// Mitsubishi GX Works2 project: Conveyor   PLC: Q03UD

PROGRAM IOCHECK
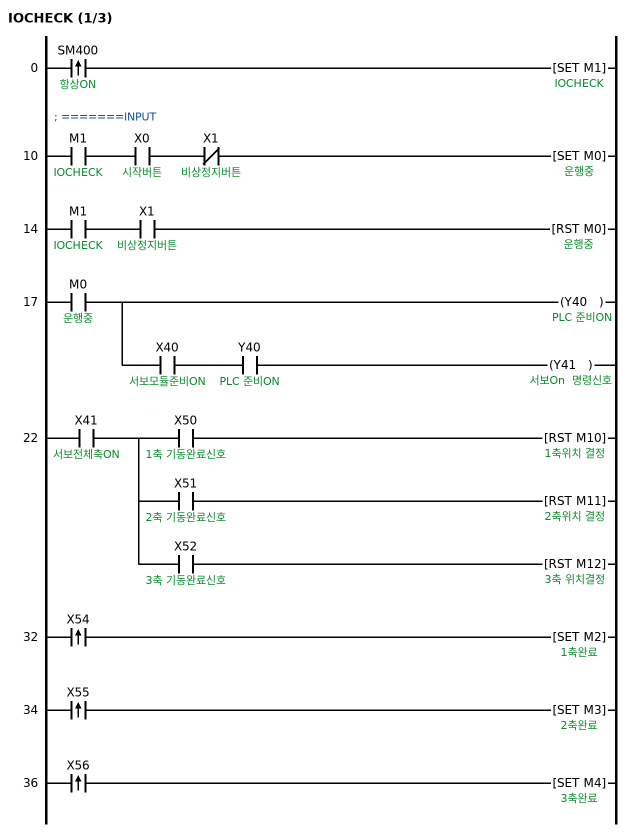
0     LDP     SM400  ; 항상ON
      SET     M1  ; IOCHECK
; =======INPUT
10    LD      M1  ; IOCHECK
      AND     X0  ; 시작버튼
      ANI     X1  ; 비상정지버튼
      SET     M0  ; 운행중
14    LD      M1  ; IOCHECK
      AND     X1  ; 비상정지버튼
      RST     M0  ; 운행중
17    LD      M0  ; 운행중
      OUT     Y40  ; PLC 준비ON
      AND     X40  ; 서보모듈준비ON
      AND     Y40  ; PLC 준비ON
      OUT     Y41  ; 서보On  명령신호
22    LD      X41  ; 서보전체축ON
      MPS
      AND     X50  ; 1축 기동완료신호
      RST     M10  ; 1축위치 결정
      MRD
      AND     X51  ; 2축 기동완료신호
      RST     M11  ; 2축위치 결정
      MPP
      AND     X52  ; 3축 기동완료신호
      RST     M12  ; 3축 위치결정
32    LDP     X54
      SET     M2  ; 1축완료
34    LDP     X55
      SET     M3  ; 2축완료
36    LDP     X56
      SET     M4  ; 3축완료
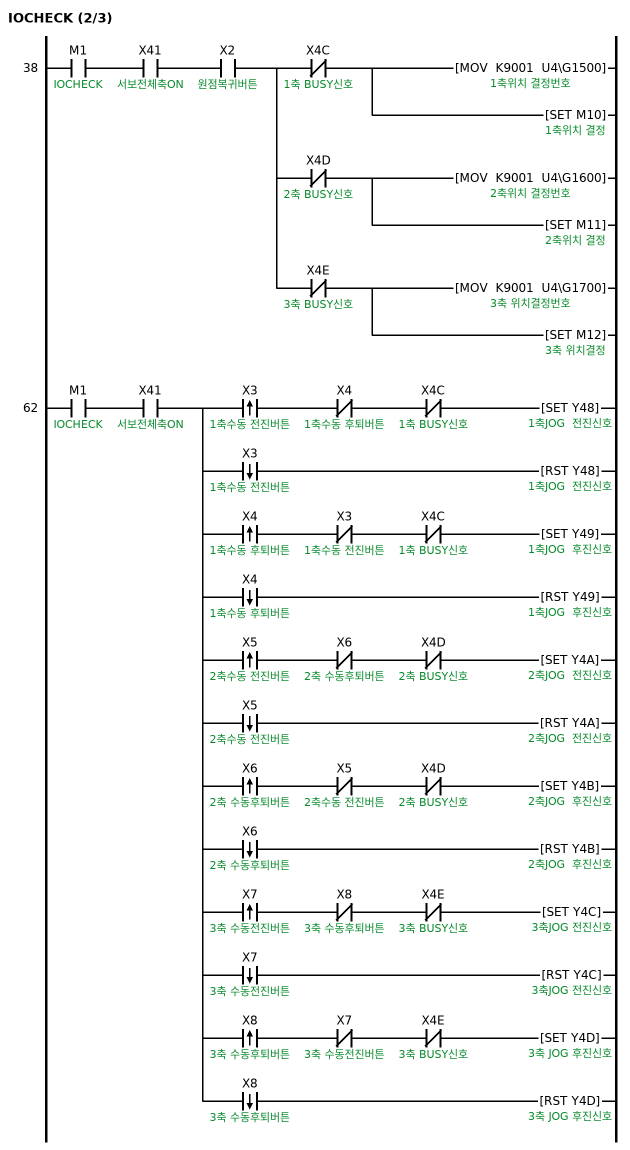
38    LD      M1  ; IOCHECK
      AND     X41  ; 서보전체축ON
      AND     X2  ; 원점복귀버튼
      MPS
      ANI     X4C  ; 1축 BUSY신호
      MOV     K9001 U4\G1500  ; 1축위치 결정번호
      SET     M10  ; 1축위치 결정
      MRD
      ANI     X4D  ; 2축 BUSY신호
      MOV     K9001 U4\G1600  ; 2축위치 결정번호
      SET     M11  ; 2축위치 결정
      MPP
      ANI     X4E  ; 3축 BUSY신호
      MOV     K9001 U4\G1700  ; 3축 위치결정번호
      SET     M12  ; 3축 위치결정
62    LD      M1  ; IOCHECK
      AND     X41  ; 서보전체축ON
      MPS
      ANDP    X3  ; 1축수동 전진버튼
      ANI     X4  ; 1축수동 후퇴버튼
      ANI     X4C  ; 1축 BUSY신호
      SET     Y48  ; 1축JOG  전진신호
      MRD
      ANDF    X3  ; 1축수동 전진버튼
      RST     Y48  ; 1축JOG  전진신호
      MRD
      ANDP    X4  ; 1축수동 후퇴버튼
      ANI     X3  ; 1축수동 전진버튼
      ANI     X4C  ; 1축 BUSY신호
      SET     Y49  ; 1축JOG  후진신호
      MRD
      ANDF    X4  ; 1축수동 후퇴버튼
      RST     Y49  ; 1축JOG  후진신호
      MRD
      ANDP    X5  ; 2축수동 전진버튼
      ANI     X6  ; 2축 수동후퇴버튼
      ANI     X4D  ; 2축 BUSY신호
      SET     Y4A  ; 2축JOG  전진신호
      MRD
      ANDF    X5  ; 2축수동 전진버튼
      RST     Y4A  ; 2축JOG  전진신호
      MRD
      ANDP    X6  ; 2축 수동후퇴버튼
      ANI     X5  ; 2축수동 전진버튼
      ANI     X4D  ; 2축 BUSY신호
      SET     Y4B  ; 2축JOG  후진신호
      MRD
      ANDF    X6  ; 2축 수동후퇴버튼
      RST     Y4B  ; 2축JOG  후진신호
      MRD
      ANDP    X7  ; 3축 수동전진버튼
      ANI     X8  ; 3축 수동후퇴버튼
      ANI     X4E  ; 3축 BUSY신호
      SET     Y4C  ; 3축JOG 전진신호
      MRD
      ANDF    X7  ; 3축 수동전진버튼
      RST     Y4C  ; 3축JOG 전진신호
      MRD
      ANDP    X8  ; 3축 수동후퇴버튼
      ANI     X7  ; 3축 수동전진버튼
      ANI     X4E  ; 3축 BUSY신호
      SET     Y4D  ; 3축 JOG 후진신호
      MPP
      ANDF    X8  ; 3축 수동후퇴버튼
      RST     Y4D  ; 3축 JOG 후진신호
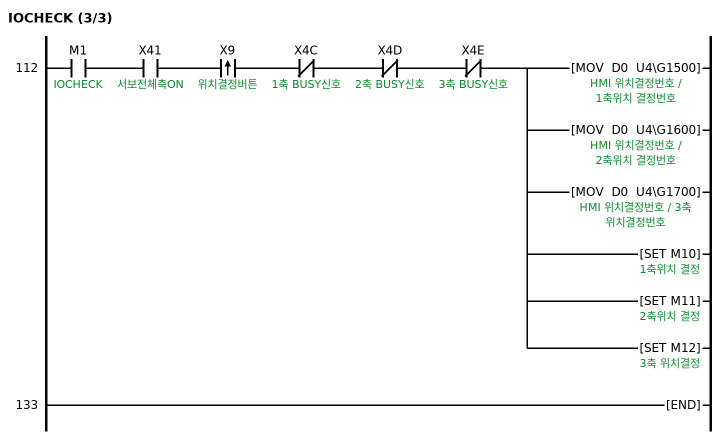
112   LD      M1  ; IOCHECK
      AND     X41  ; 서보전체축ON
      ANDP    X9  ; 위치결정버튼
      ANI     X4C  ; 1축 BUSY신호
      ANI     X4D  ; 2축 BUSY신호
      ANI     X4E  ; 3축 BUSY신호
      MOV     D0 U4\G1500  ; HMI 위치결정번호
      MOV     D0 U4\G1600
      MOV     D0 U4\G1700
      SET     M10  ; 1축위치 결정
      SET     M11  ; 2축위치 결정
      SET     M12  ; 3축 위치결정
133   END
END_PROGRAM

PROGRAM MAIN
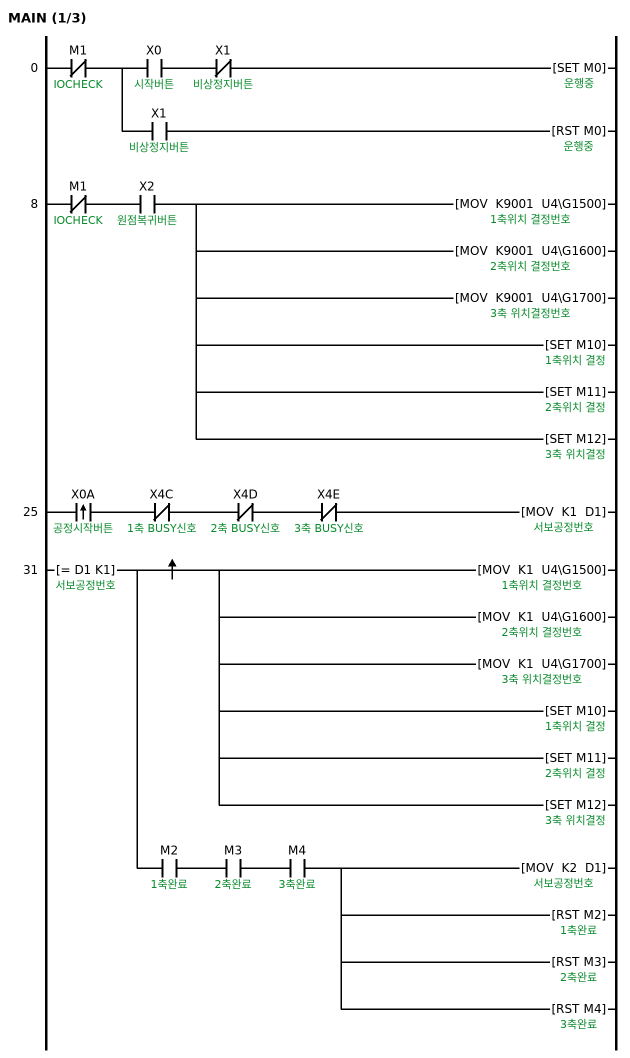
0     LDI     M1  ; IOCHECK
      MPS
      AND     X0  ; 시작버튼
      ANI     X1  ; 비상정지버튼
      SET     M0  ; 운행중
      MPP
      AND     X1  ; 비상정지버튼
      RST     M0  ; 운행중
8     LDI     M1  ; IOCHECK
      AND     X2  ; 원점복귀버튼
      MOV     K9001 U4\G1500  ; 1축위치 결정번호
      MOV     K9001 U4\G1600  ; 2축위치 결정번호
      MOV     K9001 U4\G1700  ; 3축 위치결정번호
      SET     M10  ; 1축위치 결정
      SET     M11  ; 2축위치 결정
      SET     M12  ; 3축 위치결정
25    LDP     X0A  ; 공정시작버튼
      ANI     X4C  ; 1축 BUSY신호
      ANI     X4D  ; 2축 BUSY신호
      ANI     X4E  ; 3축 BUSY신호
      MOV     K1 D1  ; 서보공정번호
31    LD=     D1 K1  ; 서보공정번호
      MPS
      MEP
      MOV     K1 U4\G1500
      MOV     K1 U4\G1600
      MOV     K1 U4\G1700
      SET     M10  ; 1축위치 결정
      SET     M11  ; 2축위치 결정
      SET     M12  ; 3축 위치결정
      MPP
      AND     M2  ; 1축완료
      AND     M3  ; 2축완료
      AND     M4  ; 3축완료
      MOV     K2 D1
      RST     M2  ; 1축완료
      RST     M3  ; 2축완료
      RST     M4  ; 3축완료
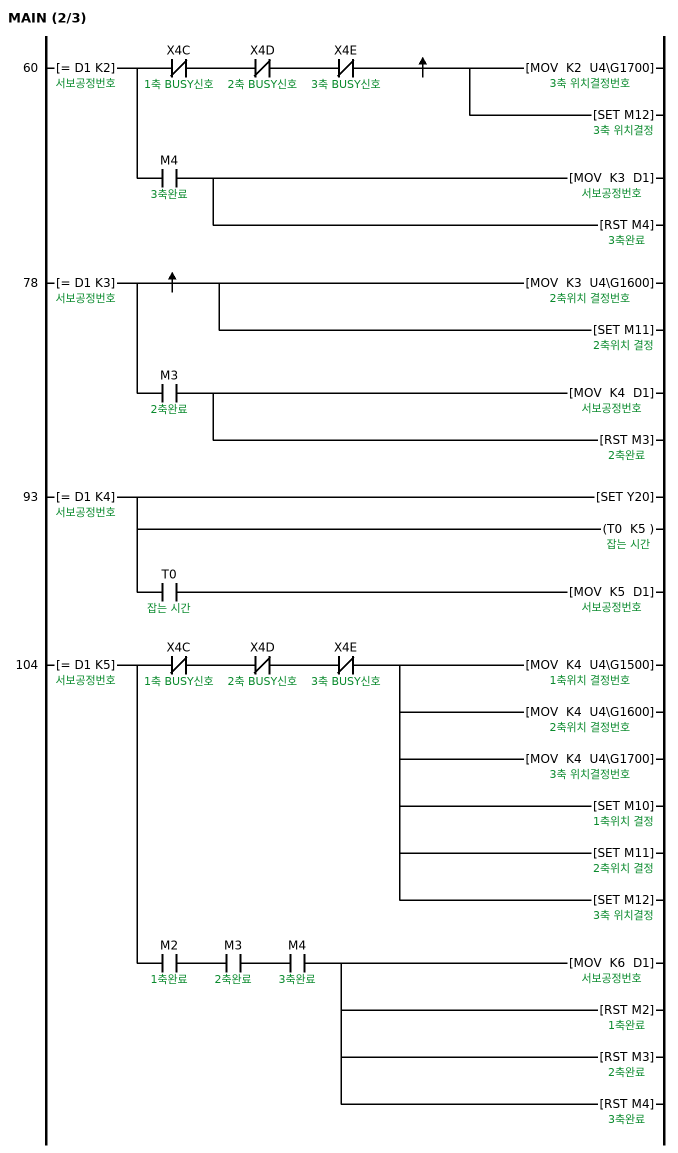
60    LD=     D1 K2  ; 서보공정번호
      MPS
      ANI     X4C  ; 1축 BUSY신호
      ANI     X4D  ; 2축 BUSY신호
      ANI     X4E  ; 3축 BUSY신호
      MEP
      MOV     K2 U4\G1700
      SET     M12  ; 3축 위치결정
      MPP
      AND     M4  ; 3축완료
      MOV     K3 D1
      RST     M4  ; 3축완료
78    LD=     D1 K3  ; 서보공정번호
      MPS
      MEP
      MOV     K3 U4\G1600
      SET     M11  ; 2축위치 결정
      MPP
      AND     M3  ; 2축완료
      MOV     K4 D1
      RST     M3  ; 2축완료
93    LD=     D1 K4  ; 서보공정번호
      SET     Y20
      OUT     T0 K5  ; 잡는 시간
      AND     T0  ; 잡는 시간
      MOV     K5 D1
104   LD=     D1 K5  ; 서보공정번호
      MPS
      ANI     X4C  ; 1축 BUSY신호
      ANI     X4D  ; 2축 BUSY신호
      ANI     X4E  ; 3축 BUSY신호
      MOV     K4 U4\G1500
      MOV     K4 U4\G1600
      MOV     K4 U4\G1700
      SET     M10  ; 1축위치 결정
      SET     M11  ; 2축위치 결정
      SET     M12  ; 3축 위치결정
      MPP
      AND     M2  ; 1축완료
      AND     M3  ; 2축완료
      AND     M4  ; 3축완료
      MOV     K6 D1
      RST     M2  ; 1축완료
      RST     M3  ; 2축완료
      RST     M4  ; 3축완료
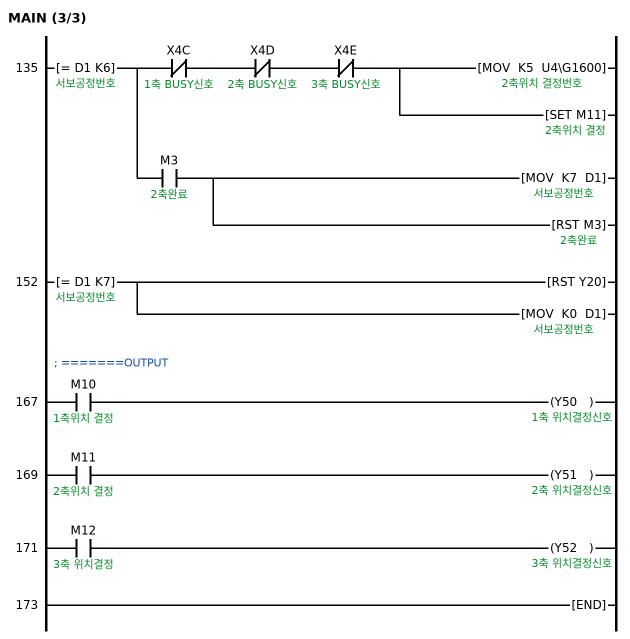
135   LD=     D1 K6  ; 서보공정번호
      MPS
      ANI     X4C  ; 1축 BUSY신호
      ANI     X4D  ; 2축 BUSY신호
      ANI     X4E  ; 3축 BUSY신호
      MOV     K5 U4\G1600
      SET     M11  ; 2축위치 결정
      MPP
      AND     M3  ; 2축완료
      MOV     K7 D1
      RST     M3  ; 2축완료
152   LD=     D1 K7  ; 서보공정번호
      RST     Y20
      MOV     K0 D1
; =======OUTPUT
167   LD      M10  ; 1축위치 결정
      OUT     Y50  ; 1축 위치결정신호
169   LD      M11  ; 2축위치 결정
      OUT     Y51  ; 2축 위치결정신호
171   LD      M12  ; 3축 위치결정
      OUT     Y52  ; 3축 위치결정신호
173   END
END_PROGRAM

PROGRAM MAIN1
0     END
END_PROGRAM
